# EPICS autosave request: leybold/centerN_settings.req
$(P):CORRFACTOR1
$(P):CORRFACTOR2
$(P):CORRFACTOR3
$(P):ERRORRELAY
$(P):FILTER1
$(P):FILTER2
$(P):FILTER3
$(P):GAS1
$(P):GAS2
$(P):GAS3
$(P):HIGHVACUUM1
$(P):HIGHVACUUM2
$(P):HIGHVACUUM3
$(P):OFFSETCORRMODE1
$(P):OFFSETCORRMODE2
$(P):OFFSETCORRMODE3
$(P):OFFSETCORRVALUE1
$(P):OFFSETCORRVALUE2
$(P):OFFSETCORRVALUE3
$(P):PARAMETERLOCK
$(P):RECORDERCHANNEL
$(P):RECORDERCURVELIN
$(P):RECORDERCURVELOG
$(P):RECORDERCURVEMODE
$(P):SENSORACTIVATIONMODE1
$(P):SENSORACTIVATIONMODE2
$(P):SENSORACTIVATIONMODE3
$(P):SENSORACTIVATIONVALUE1
$(P):SENSORACTIVATIONVALUE2
$(P):SENSORACTIVATIONVALUE3
$(P):SENSORDEACTIVATIONMODE1
$(P):SENSORDEACTIVATIONMODE2
$(P):SENSORDEACTIVATIONMODE3
$(P):SENSORDEACTIVATIONVALUE1
$(P):SENSORDEACTIVATIONVALUE2
$(P):SENSORDEACTIVATIONVALUE3
$(P):SWITCHLOWER1
$(P):SWITCHLOWER2
$(P):SWITCHLOWER3
$(P):SWITCHLOWER4
$(P):SWITCHLOWER5
$(P):SWITCHLOWER6
$(P):SWITCHMODE1
$(P):SWITCHMODE2
$(P):SWITCHMODE3
$(P):SWITCHMODE4
$(P):SWITCHMODE5
$(P):SWITCHMODE6
$(P):SWITCHUPPER1
$(P):SWITCHUPPER2
$(P):SWITCHUPPER3
$(P):SWITCHUPPER4
$(P):SWITCHUPPER5
$(P):SWITCHUPPER6
$(P):TORRLOCK
$(P):UNITS
